FUNCTION_BLOCK FB_LightOutdoor
VAR_INPUT
	bInputPIR		:	BOOL;						//Input des Bewegungsmelders
	bInputSecLoop	:	BOOL := FALSE;				//Input für Security Loop
	tHigh			:	TIME;						//Zeit (ms) für High
END_VAR
VAR_IN_OUT
	bInputHA		:	BOOL;						//Input (HA)
//	iLightMode		:	WORD;						//LichtModus für Aussenumgebung
END_VAR
VAR_OUTPUT
	bOut			:	BOOL;
END_VAR
VAR CONSTANT
	tSec			:	TIME := T#1S;
END_VAR
VAR
	fbRtrigPIR		:	R_TRIG;
	fbFtrig			:	F_TRIG;
	bTriggerPIR		:	BOOL;
	bStateOut		:	BOOL;
	
	fbRtrigInit		:	R_TRIG;
	tpPulse			:	TP;
	
	tpPulseSec		:	TP;
	tofDelaySec		:	TOF;
END_VAR

fbRtrigInit(CLK:= bInputSecLoop, Q=> );
//tpPulse(IN := bOut, PT := tHigh);

tpPulseSec(IN := bOut, PT := tSec);
tofDelaySec(IN := bOut, PT := tSec);

IF bInputSecLoop THEN	//Dauerlicht bei Security Falls

	IF fbRtrigInit.Q THEN
		bOut	:= TRUE;
	END_IF
	
	IF NOT tpPulseSec.Q THEN
		bOut := FALSE;
	END_IF
	
	IF NOT tofDelaySec.Q THEN
		bOut := TRUE;
	END_IF	
	
	bInputHA	:=	bOut;
	
ELSE	//Normale Funktion
	bTriggerPIR	:= FALSE;

	//INIT PIR TRIGGER	
	fbRtrigPIR(CLK:= bInputPIR, Q=> );
	bTriggerPIR := bTriggerPIR OR fbRtrigPIR.Q;

	// Pulse
	tpPulse(IN := bTriggerPIR, PT := tHigh);

	IF tpPulse.Q THEN
		bStateOut	:= TRUE;
	ELSIF NOT bInputHA THEN
		bStateOut 	:= FALSE;
	END_IF
	
	// Wenn über HA dauer an
	IF bInputHA THEN
		bStateOut	:= TRUE;
	END_IF
	
	fbFtrig(CLK:= bInputHA, Q=> );
	
	IF	fbFtrig.Q THEN
		bStateOut	:= FALSE;
	END_IF
	
	bOut	:= 	bStateOut;	
	
END_IF

END_FUNCTION_BLOCK

(* stored: Version 1.1.0.1, ProductVersion 3.1.4024.4
   POU FB_LightOutdoor: Id {cbbe7e41-8b68-42de-afac-9168fd20c377}, SpecialFunc None *)
